// TIA Portal V17 export
// export: Created 2026-05-13T16:54:41.3226111Z, ExportSetting WithDefaults, DisplayName Totally Integrated Automation Portal, DisplayVersion V17 Update 4, DisplayName TIA Portal Openness, DisplayVersion V17 Update 4, DisplayName TIA Portal Version Control Interface, DisplayVersion V17, DisplayName SINAMICS Startdrive Advanced, DisplayVersion V17, DisplayName SINAMICS Startdrive G130, G150, S120, S150, SINAMICS MV, S210, DisplayVersion V17, DisplayName SINAMICS Startdrive G110M, G120, G120C, G120D, G120P, G115D, DisplayVersion V17, DisplayName STEP 7 Professional, DisplayVersion V17 Update 4, DisplayName STEP 7 Safety, DisplayVersion V17, DisplayName WinCC Professional, DisplayVersion V17 Update 4
TagTable "默认变量表"
  报警字 : Word  (%MW20, HMI_连接_1, 1 s)
  报警字2 : Word  (%MW22, HMI_连接_1, 1 s)
  DB4_主管道动画 : Bool  (%M704.0, HMI_连接_1, 1 s)
  报警消音 : Bool  (%M704.1, HMI_连接_1, 1 s)
  报警字3 : Word  (%MW24, HMI_连接_1, 1 s)
  报警字4 : Word  (%MW26, HMI_连接_1, 1 s)
  报警字5 : Word  (%MW28, HMI_连接_1, 1 s)
  报警字6 : Word  (%MW30, HMI_连接_1, 1 s)
  报警字7 : Word  (%MW32, HMI_连接_1, 1 s)
  报警字8 : Word  (%MW34, HMI_连接_1, 1 s)
  报警字9 : Word  (%MW36, HMI_连接_1, 1 s)
  报警字10 : Word  (%MW38, HMI_连接_1, 1 s)
  报警字11 : Word  (%MW40, HMI_连接_1, 1 s)
  报警字12 : Word  (%MW42, HMI_连接_1, 1 s)
  自动运行报警 : Bool  (PLC tag 自动运行报警, %M844.0, HMI_连接_1, 1 s)
  自动停止 : Bool  (PLC tag 自动停止, %M844.1, HMI_连接_1, 1 s)
  A报警 : Word  (PLC tag "6-ALLALARM_DB".报警列表1.报警, HMI_连接_1, 1 s)
  A报警文本 : Array [0..15] of WString  (PLC tag "6-ALLALARM_DB".报警列表1.报警文本, HMI_连接_1, 1 s)
    TagArrayMember "[0]"
    TagArrayMember "[1]"
    TagArrayMember "[2]"
    TagArrayMember "[3]"
    TagArrayMember "[4]"
    TagArrayMember "[5]"
    TagArrayMember "[6]"
    TagArrayMember "[7]"
    TagArrayMember "[8]"
    TagArrayMember "[9]"
    TagArrayMember "[10]"
    TagArrayMember "[11]"
    TagArrayMember "[12]"
    TagArrayMember "[13]"
    TagArrayMember "[14]"
    TagArrayMember "[15]"
  B报警 : Word  (PLC tag "6-ALLALARM_DB".报警列表2.报警, HMI_连接_1, 1 s)
  B报警文本 : Array [0..15] of WString  (PLC tag "6-ALLALARM_DB".报警列表2.报警文本, HMI_连接_1, 1 s)
    TagArrayMember "[0]"
    TagArrayMember "[1]"
    TagArrayMember "[2]"
    TagArrayMember "[3]"
    TagArrayMember "[4]"
    TagArrayMember "[5]"
    TagArrayMember "[6]"
    TagArrayMember "[7]"
    TagArrayMember "[8]"
    TagArrayMember "[9]"
    TagArrayMember "[10]"
    TagArrayMember "[11]"
    TagArrayMember "[12]"
    TagArrayMember "[13]"
    TagArrayMember "[14]"
    TagArrayMember "[15]"
  C报警 : Word  (PLC tag "6-ALLALARM_DB".报警列表3.报警, HMI_连接_1, 1 s)
  C报警文本 : Array [0..15] of WString  (PLC tag "6-ALLALARM_DB".报警列表3.报警文本, HMI_连接_1, 1 s)
    TagArrayMember "[0]"
    TagArrayMember "[1]"
    TagArrayMember "[2]"
    TagArrayMember "[3]"
    TagArrayMember "[4]"
    TagArrayMember "[5]"
    TagArrayMember "[6]"
    TagArrayMember "[7]"
    TagArrayMember "[8]"
    TagArrayMember "[9]"
    TagArrayMember "[10]"
    TagArrayMember "[11]"
    TagArrayMember "[12]"
    TagArrayMember "[13]"
    TagArrayMember "[14]"
    TagArrayMember "[15]"
  D报警 : Word  (PLC tag "6-ALLALARM_DB".报警列表4.报警, HMI_连接_1, 1 s)
  D报警文本 : Array [0..15] of WString  (PLC tag "6-ALLALARM_DB".报警列表4.报警文本, HMI_连接_1, 1 s)
    TagArrayMember "[0]"
    TagArrayMember "[1]"
    TagArrayMember "[2]"
    TagArrayMember "[3]"
    TagArrayMember "[4]"
    TagArrayMember "[5]"
    TagArrayMember "[6]"
    TagArrayMember "[7]"
    TagArrayMember "[8]"
    TagArrayMember "[9]"
    TagArrayMember "[10]"
    TagArrayMember "[11]"
    TagArrayMember "[12]"
    TagArrayMember "[13]"
    TagArrayMember "[14]"
    TagArrayMember "[15]"
  E报警 : Word  (PLC tag "6-ALLALARM_DB".报警列表5.报警, HMI_连接_1, 1 s)
  E报警文本 : Array [0..15] of WString  (PLC tag "6-ALLALARM_DB".报警列表5.报警文本, HMI_连接_1, 1 s)
    TagArrayMember "[0]"
    TagArrayMember "[1]"
    TagArrayMember "[2]"
    TagArrayMember "[3]"
    TagArrayMember "[4]"
    TagArrayMember "[5]"
    TagArrayMember "[6]"
    TagArrayMember "[7]"
    TagArrayMember "[8]"
    TagArrayMember "[9]"
    TagArrayMember "[10]"
    TagArrayMember "[11]"
    TagArrayMember "[12]"
    TagArrayMember "[13]"
    TagArrayMember "[14]"
    TagArrayMember "[15]"
  F报警 : Word  (PLC tag "6-ALLALARM_DB".报警列表6.报警, HMI_连接_1, 1 s)
  F报警文本 : Array [0..15] of WString  (PLC tag "6-ALLALARM_DB".报警列表6.报警文本, HMI_连接_1, 1 s)
    TagArrayMember "[0]"
    TagArrayMember "[1]"
    TagArrayMember "[2]"
    TagArrayMember "[3]"
    TagArrayMember "[4]"
    TagArrayMember "[5]"
    TagArrayMember "[6]"
    TagArrayMember "[7]"
    TagArrayMember "[8]"
    TagArrayMember "[9]"
    TagArrayMember "[10]"
    TagArrayMember "[11]"
    TagArrayMember "[12]"
    TagArrayMember "[13]"
    TagArrayMember "[14]"
    TagArrayMember "[15]"
  G报警 : Word  (PLC tag "6-ALLALARM_DB".报警列表7.报警, HMI_连接_1, 1 s)
  G报警文本 : Array [0..15] of WString  (PLC tag "6-ALLALARM_DB".报警列表7.报警文本, HMI_连接_1, 1 s)
    TagArrayMember "[0]"
    TagArrayMember "[1]"
    TagArrayMember "[2]"
    TagArrayMember "[3]"
    TagArrayMember "[4]"
    TagArrayMember "[5]"
    TagArrayMember "[6]"
    TagArrayMember "[7]"
    TagArrayMember "[8]"
    TagArrayMember "[9]"
    TagArrayMember "[10]"
    TagArrayMember "[11]"
    TagArrayMember "[12]"
    TagArrayMember "[13]"
    TagArrayMember "[14]"
    TagArrayMember "[15]"
  H报警 : Word  (PLC tag "6-ALLALARM_DB".报警列表8.报警, HMI_连接_1, 1 s)
  H报警文本 : Array [0..15] of WString  (PLC tag "6-ALLALARM_DB".报警列表8.报警文本, HMI_连接_1, 1 s)
    TagArrayMember "[0]"
    TagArrayMember "[1]"
    TagArrayMember "[2]"
    TagArrayMember "[3]"
    TagArrayMember "[4]"
    TagArrayMember "[5]"
    TagArrayMember "[6]"
    TagArrayMember "[7]"
    TagArrayMember "[8]"
    TagArrayMember "[9]"
    TagArrayMember "[10]"
    TagArrayMember "[11]"
    TagArrayMember "[12]"
    TagArrayMember "[13]"
    TagArrayMember "[14]"
    TagArrayMember "[15]"
  I报警 : Word  (PLC tag "6-ALLALARM_DB".报警列表9.报警, HMI_连接_1, 1 s)
  I报警文本 : Array [0..15] of WString  (PLC tag "6-ALLALARM_DB".报警列表9.报警文本, HMI_连接_1, 1 s)
    TagArrayMember "[0]"
    TagArrayMember "[1]"
    TagArrayMember "[2]"
    TagArrayMember "[3]"
    TagArrayMember "[4]"
    TagArrayMember "[5]"
    TagArrayMember "[6]"
    TagArrayMember "[7]"
    TagArrayMember "[8]"
    TagArrayMember "[9]"
    TagArrayMember "[10]"
    TagArrayMember "[11]"
    TagArrayMember "[12]"
    TagArrayMember "[13]"
    TagArrayMember "[14]"
    TagArrayMember "[15]"
